TYPE "CTrk_Item"
VERSION : 0.1
// Block: CTrk_Item
   STRUCT
      C_ID : DInt;
      DecoilerX : SInt;
      MES_CN : DInt;
      MES_HN : DInt;
      Provino_Req : SInt;
      Provino_Done : SInt;
      Loaded : CTrk_Log;
      Processing : Array[1..20] of CTrk_Log;
      Consumed : CTrk_Log;
      Interrupted : CTrk_Log;
   END_STRUCT;

END_TYPE
